// Settings for GreenMaster
TYPE GreenMasterSettingsCTH2 :
STRUCT
	P2_TEMP_LIM_V: REAL := 12;
	NIGHT_COOL_EN: BOOL := FALSE; // Night cooling activation
	NIGHT_COOL_SP: REAL := 18.0; // Night cooling temperature Set Point, C
	WD_EN: BOOL := FALSE; // Watchdog enable - enables unit on watchdog update failure 
	WD_V: INT := 0; // Watchdog counter to be changed at a minimum every 5 minutes (when enabled)  
END_STRUCT
END_TYPE

(* stored: Version 1.1.0.1, ProductVersion 3.1.4024.6
   DUT GreenMasterSettingsCTH2: Id {8d674c3b-432a-4cf2-9ffd-5b24fccd3039} *)
